// TwinCAT 3 PLC project txi_hxr_optics
// Title: lcls-plc-txi-hxr-optics
// Company: SLAC
// ProjectVersion: 1.0.0
// ProgramVersion: 3.1.4022.7
// libraries:
//   lcls-twincat-motion, * (SLAC)
//   lcls-twincat-optics, * (SLAC)
//   PMPS, * (SLAC - LCLS)
//   Tc2_Standard, * (Beckhoff Automation GmbH)
//   Tc2_System, * (Beckhoff Automation GmbH)
//   Tc3_Module, * (Beckhoff Automation GmbH)
// project tree:
//   GVLs/ GVL_MR1L1_Constants.TcGVL, GVL_PMPS.TcGVL, Main.TcGVL
//   Version/ Global_Version.TcGVL
//   / PlcTask.TcTTO
//   POUs/ PRG_1_PlcTask.TcPOU, PRG_2_PMPS_POST.TcPOU, PRG_MR1L1_HOMS.TcPOU
// real-time tasks:
//   TASK PlcTask: cycle T#10ms, priority 20, ADS port 350
// motion (NC):
//   TASK NC-Task 1 SAF: cycle T#2ms, priority 4, ADS port 501
//   TASK NC-Task 1 SVB: cycle T#10ms, priority 8, ADS port 511
//   AXIS Axis 1 MR1L1-HOMS-YUP (id 1)
//     General: UnitName=um
//     Dynamic: Acceleration=5050, Deceleration=5050, Jerk=5100500, DelayTime=0.008
//     Velo: SlowManual=60, FastManual=90, Maximum=500
//     OtherSettings: AllowMotionCmdToSlave=true
//     encoder EncType=29
//       EncPara: ScaleFactorNumerator=1, ScaleFactorDenominator=1000, MaxCount=#xffffffff
//         SoftEndMaxControl: Enable=true, Range=121500
//         Inc: RefSoftSyncMask=#x0000ffff
//     drive DrvType=24
//       DrvPara: Inverse=true
//         Analog: VeloReferenz=500, ScaleFactorActTorque=0.1
//         TimeComp: TaskDelayCycles=1
//     controller CtrType=3
//       CtrPara: PriorControlFactor=1
//         PosDiffControl: Range=50, Time=0.2
//         PID: PosTn=0.005, PosIOutputLimit=0.0001, PosDOutputLimit=0, PosIDisableWhenMoving=true, DeadBandPosition=0.001
//         Observer: BandWidth=20
//   AXIS Axis 2 MR1L1-HOMS-YDWN (id 2)
//     General: UnitName=um
//     Dynamic: Acceleration=5050, Deceleration=5050, Jerk=5100500, DelayTime=0.008
//     Velo: SlowManual=60, FastManual=90, Maximum=500
//     OtherSettings: AllowMotionCmdToSlave=true
//     encoder EncType=29
//       EncPara: ScaleFactorNumerator=1, ScaleFactorDenominator=1000, MaxCount=#xffffffff
//         Inc: RefSoftSyncMask=#x0000ffff
//     drive DrvType=24
//       DrvPara: Inverse=true
//         Analog: VeloReferenz=500, ScaleFactorActTorque=0.1
//         TimeComp: TaskDelayCycles=1
//     controller CtrType=3
//       CtrPara: PriorControlFactor=1
//         PosDiffControl: Range=50, Time=0.2
//         PID: PosTn=0.005, PosIOutputLimit=0.0001, PosDOutputLimit=0, PosIDisableWhenMoving=true, DeadBandPosition=0.001
//         Observer: BandWidth=20
//   AXIS Axis 3 MR1L1-HOMS-XUP (id 3)
//     General: UnitName=um
//     Dynamic: Acceleration=1000, Deceleration=1000, Jerk=5000, DelayTime=0.008
//     Velo: FastManual=150, Maximum=150
//     OtherSettings: AllowMotionCmdToSlave=true
//     encoder EncType=29
//       EncPara: ScaleFactorNumerator=0.001, MaxCount=#xffffffff
//         Inc: RefSoftSyncMask=#x0000ffff
//     drive DrvType=24
//       DrvPara: Inverse=true
//         Analog: VeloReferenz=625, ScaleFactorActTorque=0.1
//         TimeComp: TaskDelayCycles=1
//     controller CtrType=1
//       CtrPara: PriorControlFactor=1
//         PosDiffControl: Range=50
//         Observer: BandWidth=20
//   AXIS Axis 4 MR1L1-HOMS-XDWN (id 4)
//     General: UnitName=um
//     Dynamic: Acceleration=1000, Deceleration=1000, Jerk=5000, DelayTime=0.008
//     Velo: FastManual=150, Maximum=150
//     OtherSettings: AllowMotionCmdToSlave=true
//     encoder EncType=29
//       EncPara: ScaleFactorNumerator=0.001, MaxCount=#xffffffff
//         Inc: RefSoftSyncMask=#x0000ffff
//     drive DrvType=24
//       Analog: VeloReferenz=625, ScaleFactorActTorque=0.1
//       TimeComp: TaskDelayCycles=1
//     controller CtrType=1
//       CtrPara: PriorControlFactor=1
//         PosDiffControl: Range=50
//         Observer: BandWidth=20
//   AXIS Axis 5 MR1L1-HOMS-PITCH (id 5)
//     General: UnitName=urad
//     Dynamic: AccelerationMaximum=7042, Acceleration=7000, Deceleration=14000, DelayTime=0.008, VeloJumpFactor=2000
//     Velo: SlowManual=30, FastManual=50, Maximum=400
//     MotionControl: Time=0.1
//     TargetPosControl: Time=2
//     OtherSettings: AllowMotionCmdToSlave=true, AllowMotionCmdToExtSetGenAxis=true, PulseDistancePos=100
//     encoder EncType=29
//       EncPara: ScaleFactorNumerator=0.00556, MaxCount=#xffffffff
//         Inc: RefSoftSyncMask=#x0000ffff
//     drive DrvType=24
//       DrvPara: Inverse=true
//         Analog: VeloReferenz=550.176
//         TimeComp: TaskDelayCycles=1
//     controller CtrType=3
//       CtrPara: PriorControlFactor=1
//         PosDiffControl: Range=10, Time=0.2
//         PID: PosKp=8, PosTn=0.0005, PosIOutputLimit=5e-05, PosDOutputLimit=0, DeadBandPosition=0.1
//         Observer: BandWidth=20
// I/O:
//   DEVICE Device 1 (EtherCAT), AmsNetId 172.21.136.43.2.1
//     Term 1 (EK1200) [EK1200-5000 EtherCAT Power supply (2A E-Bus)]
//       PMPS_FFO
//       License (6070)
//       PMPS_PRE [EL6695 EtherCAT Bridge terminal (Primary)]
//       PLC Junction 1 (EK1122) [EK1122 2 port EtherCAT junction]
//         X1 MR1L1 (EK1100) [EK1100 EtherCAT Coupler (2A E-Bus)]
//           Term 8 (EL9410)
//           MR1L1-EL7047-E01 [EL7047 1Ch. Stepper motor output stage (50V, 5A)]
//           MR1L1-EL7047-E02 [EL7047 1Ch. Stepper motor output stage (50V, 5A)]
//           MR1L1-EL7047-E03 [EL7047 1Ch. Stepper motor output stage (50V, 5A)]
//           MR1L1-EL7047-E04 [EL7047 1Ch. Stepper motor output stage (50V, 5A)]
//           MR1L1-EL7047-E05 [EL7047 1Ch. Stepper motor output stage (50V, 5A)]
//           MR1L1-EL5042-E06 [EL5042 2Ch. BiSS-C Encoder]
//           MR1L1-EL5042-E07 [EL5042 2Ch. BiSS-C Encoder]
//           MR1L1-EL5042-E08 [EL5042 2Ch. BiSS-C Encoder]
//           MR1L1-EL6001-E09 [EL6001 Interface (RS232)]
//           MR1L1-EL3054-E10 [EL3054 4Ch. Ana. Input 4-20mA]
//           MR1L1-EL3202-0010-E11 [EL3202-0010 2Ch. Ana. Input PT100 (RTD), High Precision]
//           MR1L1-EL3202-0010-E12 [EL3202-0010 2Ch. Ana. Input PT100 (RTD), High Precision]
//           MR1L1-EL1004-E13
//           MR1L1-EL2004-E14 [EL2004 4Ch. Dig. Output 24V, 0.5A]
//           Term 19 (EL9011) [EL9011 End Terminal]
// variable links:
//   Axes/Axis 1 MR1L1-HOMS-YUP <-> Device 1 (EtherCAT)/Term 1 (EK1200)/PLC Junction 1 (EK1122)/X1 MR1L1 (EK1100)/MR1L1-EL5042-E06
//     Enc/Inputs/In/nComState @bit 1 <-> WcState/InputToggle
//     Enc/Inputs/In/nComState <-> WcState/WcState
//     Enc/Inputs/In/nDataIn1 <-> FB Inputs Channel 1/Position
//     Enc/Inputs/In/nState1 @bit 12 <-> FB Inputs Channel 1/Status/Diag
//     Enc/Inputs/In/nState1 @bit 1 <-> FB Inputs Channel 1/Status/Error
//     Enc/Inputs/In/nState1 @bit 14 <-> FB Inputs Channel 1/Status/Input cycle counter
//     Enc/Inputs/In/nState1 @bit 2 <-> FB Inputs Channel 1/Status/Ready
//     Enc/Inputs/In/nState1 @bit 13 <-> FB Inputs Channel 1/Status/TxPDO State
//     Enc/Inputs/In/nState1 <-> FB Inputs Channel 1/Status/Warning
//   Axes/Axis 1 MR1L1-HOMS-YUP <-> Device 1 (EtherCAT)/Term 1 (EK1200)/PLC Junction 1 (EK1122)/X1 MR1L1 (EK1100)/MR1L1-EL7047-E01
//     Drive/Inputs/In/nState1 @bit 3 <-> STM Status/Status/Error
//     Drive/Inputs/In/nState1 @bit 7 <-> STM Status/Status/Motor stall
//     Drive/Inputs/In/nState1 @bit 5 <-> STM Status/Status/Moving negative
//     Drive/Inputs/In/nState1 @bit 4 <-> STM Status/Status/Moving positive
//     Drive/Inputs/In/nState1 @bit 1 <-> STM Status/Status/Ready
//     Drive/Inputs/In/nState1 <-> STM Status/Status/Ready to enable
//     Drive/Inputs/In/nState1 @bit 6 <-> STM Status/Status/Torque reduced
//     Drive/Inputs/In/nState1 @bit 2 <-> STM Status/Status/Warning
//     Drive/Inputs/In/nState2 @bit 3 <-> STM Status/Status/Digital input 1
//     Drive/Inputs/In/nState2 @bit 4 <-> STM Status/Status/Digital input 2
//     Drive/Inputs/In/nState2 @bit 5 <-> STM Status/Status/Sync error
//     Drive/Inputs/In/nState2 @bit 7 <-> STM Status/Status/TxPDO Toggle
//     Drive/Inputs/In/nState4 @bit 1 <-> WcState/InputToggle
//     Drive/Inputs/In/nState4 <-> WcState/WcState
//     Drive/Outputs/Out/nCtrl1 <-> STM Control/Control/Enable
//     Drive/Outputs/Out/nCtrl1 @bit 2 <-> STM Control/Control/Reduce torque
//     Drive/Outputs/Out/nCtrl1 @bit 1 <-> STM Control/Control/Reset
//     Drive/Outputs/Out/nCtrl2 @bit 3 <-> STM Control/Control/Digital output 1
//     Drive/Outputs/Out/nDataOut2[0] <-> STM Velocity/Velocity
//   Axes/Axis 2 MR1L1-HOMS-YDWN <-> Device 1 (EtherCAT)/Term 1 (EK1200)/PLC Junction 1 (EK1122)/X1 MR1L1 (EK1100)/MR1L1-EL5042-E06
//     Enc/Inputs/In/nComState @bit 1 <-> WcState/InputToggle
//     Enc/Inputs/In/nComState <-> WcState/WcState
//     Enc/Inputs/In/nDataIn1 <-> FB Inputs Channel 2/Position
//     Enc/Inputs/In/nState1 @bit 12 <-> FB Inputs Channel 2/Status/Diag
//     Enc/Inputs/In/nState1 @bit 1 <-> FB Inputs Channel 2/Status/Error
//     Enc/Inputs/In/nState1 @bit 14 <-> FB Inputs Channel 2/Status/Input cycle counter
//     Enc/Inputs/In/nState1 @bit 2 <-> FB Inputs Channel 2/Status/Ready
//     Enc/Inputs/In/nState1 @bit 13 <-> FB Inputs Channel 2/Status/TxPDO State
//     Enc/Inputs/In/nState1 <-> FB Inputs Channel 2/Status/Warning
//   Axes/Axis 2 MR1L1-HOMS-YDWN <-> Device 1 (EtherCAT)/Term 1 (EK1200)/PLC Junction 1 (EK1122)/X1 MR1L1 (EK1100)/MR1L1-EL7047-E02
//     Drive/Inputs/In/nState1 @bit 3 <-> STM Status/Status/Error
//     Drive/Inputs/In/nState1 @bit 7 <-> STM Status/Status/Motor stall
//     Drive/Inputs/In/nState1 @bit 5 <-> STM Status/Status/Moving negative
//     Drive/Inputs/In/nState1 @bit 4 <-> STM Status/Status/Moving positive
//     Drive/Inputs/In/nState1 @bit 1 <-> STM Status/Status/Ready
//     Drive/Inputs/In/nState1 <-> STM Status/Status/Ready to enable
//     Drive/Inputs/In/nState1 @bit 6 <-> STM Status/Status/Torque reduced
//     Drive/Inputs/In/nState1 @bit 2 <-> STM Status/Status/Warning
//     Drive/Inputs/In/nState2 @bit 3 <-> STM Status/Status/Digital input 1
//     Drive/Inputs/In/nState2 @bit 4 <-> STM Status/Status/Digital input 2
//     Drive/Inputs/In/nState2 @bit 5 <-> STM Status/Status/Sync error
//     Drive/Inputs/In/nState2 @bit 7 <-> STM Status/Status/TxPDO Toggle
//     Drive/Inputs/In/nState4 @bit 1 <-> WcState/InputToggle
//     Drive/Inputs/In/nState4 <-> WcState/WcState
//     Drive/Outputs/Out/nCtrl1 <-> STM Control/Control/Enable
//     Drive/Outputs/Out/nCtrl1 @bit 2 <-> STM Control/Control/Reduce torque
//     Drive/Outputs/Out/nCtrl1 @bit 1 <-> STM Control/Control/Reset
//     Drive/Outputs/Out/nCtrl2 @bit 3 <-> STM Control/Control/Digital output 1
//     Drive/Outputs/Out/nDataOut2[0] <-> STM Velocity/Velocity
//   Axes/Axis 3 MR1L1-HOMS-XUP <-> Device 1 (EtherCAT)/Term 1 (EK1200)/PLC Junction 1 (EK1122)/X1 MR1L1 (EK1100)/MR1L1-EL5042-E07
//     Enc/Inputs/In/nComState @bit 1 <-> WcState/InputToggle
//     Enc/Inputs/In/nComState <-> WcState/WcState
//     Enc/Inputs/In/nDataIn1 <-> FB Inputs Channel 1/Position
//     Enc/Inputs/In/nState1 @bit 12 <-> FB Inputs Channel 1/Status/Diag
//     Enc/Inputs/In/nState1 @bit 1 <-> FB Inputs Channel 1/Status/Error
//     Enc/Inputs/In/nState1 @bit 14 <-> FB Inputs Channel 1/Status/Input cycle counter
//     Enc/Inputs/In/nState1 @bit 2 <-> FB Inputs Channel 1/Status/Ready
//     Enc/Inputs/In/nState1 @bit 13 <-> FB Inputs Channel 1/Status/TxPDO State
//     Enc/Inputs/In/nState1 <-> FB Inputs Channel 1/Status/Warning
//   Axes/Axis 3 MR1L1-HOMS-XUP <-> Device 1 (EtherCAT)/Term 1 (EK1200)/PLC Junction 1 (EK1122)/X1 MR1L1 (EK1100)/MR1L1-EL7047-E03
//     Drive/Inputs/In/nState1 @bit 3 <-> STM Status/Status/Error
//     Drive/Inputs/In/nState1 @bit 7 <-> STM Status/Status/Motor stall
//     Drive/Inputs/In/nState1 @bit 5 <-> STM Status/Status/Moving negative
//     Drive/Inputs/In/nState1 @bit 4 <-> STM Status/Status/Moving positive
//     Drive/Inputs/In/nState1 @bit 1 <-> STM Status/Status/Ready
//     Drive/Inputs/In/nState1 <-> STM Status/Status/Ready to enable
//     Drive/Inputs/In/nState1 @bit 6 <-> STM Status/Status/Torque reduced
//     Drive/Inputs/In/nState1 @bit 2 <-> STM Status/Status/Warning
//     Drive/Inputs/In/nState2 @bit 3 <-> STM Status/Status/Digital input 1
//     Drive/Inputs/In/nState2 @bit 4 <-> STM Status/Status/Digital input 2
//     Drive/Inputs/In/nState2 @bit 5 <-> STM Status/Status/Sync error
//     Drive/Inputs/In/nState2 @bit 7 <-> STM Status/Status/TxPDO Toggle
//     Drive/Inputs/In/nState4 @bit 1 <-> WcState/InputToggle
//     Drive/Inputs/In/nState4 <-> WcState/WcState
//     Drive/Outputs/Out/nCtrl1 <-> STM Control/Control/Enable
//     Drive/Outputs/Out/nCtrl1 @bit 2 <-> STM Control/Control/Reduce torque
//     Drive/Outputs/Out/nCtrl1 @bit 1 <-> STM Control/Control/Reset
//     Drive/Outputs/Out/nCtrl2 @bit 3 <-> STM Control/Control/Digital output 1
//     Drive/Outputs/Out/nDataOut2[0] <-> STM Velocity/Velocity
//   Axes/Axis 4 MR1L1-HOMS-XDWN <-> Device 1 (EtherCAT)/Term 1 (EK1200)/PLC Junction 1 (EK1122)/X1 MR1L1 (EK1100)/MR1L1-EL5042-E07
//     Enc/Inputs/In/nComState @bit 1 <-> WcState/InputToggle
//     Enc/Inputs/In/nComState <-> WcState/WcState
//     Enc/Inputs/In/nDataIn1 <-> FB Inputs Channel 2/Position
//     Enc/Inputs/In/nState1 @bit 12 <-> FB Inputs Channel 2/Status/Diag
//     Enc/Inputs/In/nState1 @bit 1 <-> FB Inputs Channel 2/Status/Error
//     Enc/Inputs/In/nState1 @bit 14 <-> FB Inputs Channel 2/Status/Input cycle counter
//     Enc/Inputs/In/nState1 @bit 2 <-> FB Inputs Channel 2/Status/Ready
//     Enc/Inputs/In/nState1 @bit 13 <-> FB Inputs Channel 2/Status/TxPDO State
//     Enc/Inputs/In/nState1 <-> FB Inputs Channel 2/Status/Warning
//   Axes/Axis 4 MR1L1-HOMS-XDWN <-> Device 1 (EtherCAT)/Term 1 (EK1200)/PLC Junction 1 (EK1122)/X1 MR1L1 (EK1100)/MR1L1-EL7047-E04
//     Drive/Inputs/In/nState1 @bit 3 <-> STM Status/Status/Error
//     Drive/Inputs/In/nState1 @bit 7 <-> STM Status/Status/Motor stall
//     Drive/Inputs/In/nState1 @bit 5 <-> STM Status/Status/Moving negative
//     Drive/Inputs/In/nState1 @bit 4 <-> STM Status/Status/Moving positive
//     Drive/Inputs/In/nState1 @bit 1 <-> STM Status/Status/Ready
//     Drive/Inputs/In/nState1 <-> STM Status/Status/Ready to enable
//     Drive/Inputs/In/nState1 @bit 6 <-> STM Status/Status/Torque reduced
//     Drive/Inputs/In/nState1 @bit 2 <-> STM Status/Status/Warning
//     Drive/Inputs/In/nState2 @bit 3 <-> STM Status/Status/Digital input 1
//     Drive/Inputs/In/nState2 @bit 4 <-> STM Status/Status/Digital input 2
//     Drive/Inputs/In/nState2 @bit 5 <-> STM Status/Status/Sync error
//     Drive/Inputs/In/nState2 @bit 7 <-> STM Status/Status/TxPDO Toggle
//     Drive/Inputs/In/nState4 @bit 1 <-> WcState/InputToggle
//     Drive/Inputs/In/nState4 <-> WcState/WcState
//     Drive/Outputs/Out/nCtrl1 <-> STM Control/Control/Enable
//     Drive/Outputs/Out/nCtrl1 @bit 2 <-> STM Control/Control/Reduce torque
//     Drive/Outputs/Out/nCtrl1 @bit 1 <-> STM Control/Control/Reset
//     Drive/Outputs/Out/nCtrl2 @bit 3 <-> STM Control/Control/Digital output 1
//     Drive/Outputs/Out/nDataOut2[0] <-> STM Velocity/Velocity
//   Axes/Axis 5 MR1L1-HOMS-PITCH <-> Device 1 (EtherCAT)/Term 1 (EK1200)/PLC Junction 1 (EK1122)/X1 MR1L1 (EK1100)/MR1L1-EL5042-E08
//     Enc/Inputs/In/nComState @bit 1 <-> WcState/InputToggle
//     Enc/Inputs/In/nComState <-> WcState/WcState
//     Enc/Inputs/In/nDataIn1 <-> FB Inputs Channel 1/Position
//     Enc/Inputs/In/nState1 @bit 12 <-> FB Inputs Channel 1/Status/Diag
//     Enc/Inputs/In/nState1 @bit 1 <-> FB Inputs Channel 1/Status/Error
//     Enc/Inputs/In/nState1 @bit 14 <-> FB Inputs Channel 1/Status/Input cycle counter
//     Enc/Inputs/In/nState1 @bit 2 <-> FB Inputs Channel 1/Status/Ready
//     Enc/Inputs/In/nState1 @bit 13 <-> FB Inputs Channel 1/Status/TxPDO State
//     Enc/Inputs/In/nState1 <-> FB Inputs Channel 1/Status/Warning
//   Axes/Axis 5 MR1L1-HOMS-PITCH <-> Device 1 (EtherCAT)/Term 1 (EK1200)/PLC Junction 1 (EK1122)/X1 MR1L1 (EK1100)/MR1L1-EL7047-E05
//     Drive/Inputs/In/nState1 @bit 3 <-> STM Status/Status/Error
//     Drive/Inputs/In/nState1 @bit 7 <-> STM Status/Status/Motor stall
//     Drive/Inputs/In/nState1 @bit 5 <-> STM Status/Status/Moving negative
//     Drive/Inputs/In/nState1 @bit 4 <-> STM Status/Status/Moving positive
//     Drive/Inputs/In/nState1 @bit 1 <-> STM Status/Status/Ready
//     Drive/Inputs/In/nState1 <-> STM Status/Status/Ready to enable
//     Drive/Inputs/In/nState1 @bit 6 <-> STM Status/Status/Torque reduced
//     Drive/Inputs/In/nState1 @bit 2 <-> STM Status/Status/Warning
//     Drive/Inputs/In/nState2 @bit 3 <-> STM Status/Status/Digital input 1
//     Drive/Inputs/In/nState2 @bit 4 <-> STM Status/Status/Digital input 2
//     Drive/Inputs/In/nState2 @bit 5 <-> STM Status/Status/Sync error
//     Drive/Inputs/In/nState2 @bit 7 <-> STM Status/Status/TxPDO Toggle
//     Drive/Inputs/In/nState4 @bit 1 <-> WcState/InputToggle
//     Drive/Inputs/In/nState4 <-> WcState/WcState
//     Drive/Outputs/Out/nCtrl1 <-> STM Control/Control/Enable
//     Drive/Outputs/Out/nCtrl1 @bit 2 <-> STM Control/Control/Reduce torque
//     Drive/Outputs/Out/nCtrl1 @bit 1 <-> STM Control/Control/Reset
//     Drive/Outputs/Out/nCtrl2 @bit 3 <-> STM Control/Control/Digital output 1
//     Drive/Outputs/Out/nDataOut2[0] <-> STM Velocity/Velocity
//   txi_hxr_optics Instance <-> Device 1 (EtherCAT)/Term 1 (EK1200)/PLC Junction 1 (EK1122)/X1 MR1L1 (EK1100)/MR1L1-EL1004-E13
//     PlcTask Inputs/PRG_MR1L1_HOMS.MR1L1.fbRunHOMS.bSTOEnable1 <-> Channel 1/Input
//     PlcTask Inputs/PRG_MR1L1_HOMS.MR1L1.fbRunHOMS.bSTOEnable2 <-> Channel 2/Input
//   txi_hxr_optics Instance <-> Device 1 (EtherCAT)/Term 1 (EK1200)/PLC Junction 1 (EK1122)/X1 MR1L1 (EK1100)/MR1L1-EL2004-E14
//     PlcTask Outputs/PRG_MR1L1_HOMS.bActivateVarCool <-> Channel 1/Output
//   txi_hxr_optics Instance <-> Device 1 (EtherCAT)/Term 1 (EK1200)/PLC Junction 1 (EK1122)/X1 MR1L1 (EK1100)/MR1L1-EL3054-E10
//     PlcTask Inputs/PRG_MR1L1_HOMS.fbCoolingPanel.fbFlow_1.iRaw <-> AI Standard Channel 1/Value
//     PlcTask Inputs/PRG_MR1L1_HOMS.fbCoolingPanel.fbFlow_2.iRaw <-> AI Standard Channel 2/Value
//     PlcTask Inputs/PRG_MR1L1_HOMS.fbCoolingPanel.fbPress_1.iRaw <-> AI Standard Channel 3/Value
//   txi_hxr_optics Instance <-> Device 1 (EtherCAT)/Term 1 (EK1200)/PLC Junction 1 (EK1122)/X1 MR1L1 (EK1100)/MR1L1-EL5042-E06
//     PlcTask Inputs/Main.M1.nRawEncoderULINT <-> FB Inputs Channel 1/Position
//     PlcTask Inputs/Main.M2.nRawEncoderULINT <-> FB Inputs Channel 2/Position
//     PlcTask Inputs/PRG_MR1L1_HOMS.MR1L1.fbRunHOMS.stYdwnEnc/Count <-> FB Inputs Channel 2/Position
//     PlcTask Inputs/PRG_MR1L1_HOMS.MR1L1.fbRunHOMS.stYupEnc/Count <-> FB Inputs Channel 1/Position
//     PlcTask Inputs/PRG_MR1L1_HOMS.bMR1L1_Y_ENC_Ready <-> FB Inputs Channel 1/Status/Ready
//     PlcTask Inputs/PRG_MR1L1_HOMS.bMR1L1_Y_ENC_TxPDO <-> FB Inputs Channel 1/Status/TxPDO State
//   txi_hxr_optics Instance <-> Device 1 (EtherCAT)/Term 1 (EK1200)/PLC Junction 1 (EK1122)/X1 MR1L1 (EK1100)/MR1L1-EL5042-E07
//     PlcTask Inputs/Main.M3.nRawEncoderULINT <-> FB Inputs Channel 1/Position
//     PlcTask Inputs/Main.M4.nRawEncoderULINT <-> FB Inputs Channel 2/Position
//     PlcTask Inputs/PRG_MR1L1_HOMS.MR1L1.fbRunHOMS.stXdwnEnc/Count <-> FB Inputs Channel 2/Position
//     PlcTask Inputs/PRG_MR1L1_HOMS.MR1L1.fbRunHOMS.stXupEnc/Count <-> FB Inputs Channel 1/Position
//   txi_hxr_optics Instance <-> Device 1 (EtherCAT)/Term 1 (EK1200)/PLC Junction 1 (EK1122)/X1 MR1L1 (EK1100)/MR1L1-EL5042-E08
//     PlcTask Inputs/Main.M5.nRawEncoderULINT <-> FB Inputs Channel 1/Position
//   txi_hxr_optics Instance <-> Device 1 (EtherCAT)/Term 1 (EK1200)/PLC Junction 1 (EK1122)/X1 MR1L1 (EK1100)/MR1L1-EL7047-E01
//     PlcTask Inputs/Main.M1.bLimitBackwardEnable <-> STM Status/Status/Digital input 2
//     PlcTask Inputs/Main.M1.bLimitForwardEnable <-> STM Status/Status/Digital input 1
//   txi_hxr_optics Instance <-> Device 1 (EtherCAT)/Term 1 (EK1200)/PLC Junction 1 (EK1122)/X1 MR1L1 (EK1100)/MR1L1-EL7047-E02
//     PlcTask Inputs/Main.M2.bLimitBackwardEnable <-> STM Status/Status/Digital input 2
//     PlcTask Inputs/Main.M2.bLimitForwardEnable <-> STM Status/Status/Digital input 1
//   txi_hxr_optics Instance <-> Device 1 (EtherCAT)/Term 1 (EK1200)/PLC Junction 1 (EK1122)/X1 MR1L1 (EK1100)/MR1L1-EL7047-E03
//     PlcTask Inputs/Main.M3.bLimitBackwardEnable <-> STM Status/Status/Digital input 2
//     PlcTask Inputs/Main.M3.bLimitForwardEnable <-> STM Status/Status/Digital input 1
//   txi_hxr_optics Instance <-> Device 1 (EtherCAT)/Term 1 (EK1200)/PLC Junction 1 (EK1122)/X1 MR1L1 (EK1100)/MR1L1-EL7047-E04
//     PlcTask Inputs/Main.M4.bLimitBackwardEnable <-> STM Status/Status/Digital input 2
//     PlcTask Inputs/Main.M4.bLimitForwardEnable <-> STM Status/Status/Digital input 1
//   txi_hxr_optics Instance <-> Device 1 (EtherCAT)/Term 1 (EK1200)/PLC Junction 1 (EK1122)/X1 MR1L1 (EK1100)/MR1L1-EL7047-E05
//     PlcTask Inputs/Main.M5.bLimitBackwardEnable <-> STM Status/Status/Digital input 2
//     PlcTask Inputs/Main.M5.bLimitForwardEnable <-> STM Status/Status/Digital input 1
//   txi_hxr_optics Instance <-> Device 1 (EtherCAT)/Term 1 (EK1200)/PMPS_FFO
//     PlcTask Outputs/GVL_PMPS.fbFastFaultOutput1.q_xFastFaultOut <-> Channel 1/Output
//   txi_hxr_optics Instance <-> Device 1 (EtherCAT)/Term 1 (EK1200)/PMPS_PRE
//     PlcTask Inputs/PRG_2_PMPS_POST.fbArbiterIO.i_stCurrentBP <-> IO Inputs/CurrentBP
//     PlcTask Inputs/PRG_2_PMPS_POST.fbArbiterIO.xTxPDO_state <-> SYNC Inputs/TxPDO state
//     PlcTask Inputs/PRG_2_PMPS_POST.fbArbiterIO.xTxPDO_toggle <-> SYNC Inputs/TxPDO toggle
//     PlcTask Outputs/PRG_2_PMPS_POST.fbArbiterIO.q_stRequestedBP <-> IO Outputs/RequestedBP
//     PlcTask Outputs/PRG_MR1L1_HOMS.nMR1L1_Y_ENC_PMPS <-> IO Outputs/MR1L1_Y_ENC
//   txi_hxr_optics Instance <-> NC-Task 1 SAF/Axes/Axis 1 MR1L1-HOMS-YUP
//     PlcTask Inputs/Main.M1.Axis.NcToPlc <-> Outputs/ToPlc
//     PlcTask Outputs/Main.M1.Axis.PlcToNc <-> Inputs/FromPlc
//   txi_hxr_optics Instance <-> NC-Task 1 SAF/Axes/Axis 2 MR1L1-HOMS-YDWN
//     PlcTask Inputs/Main.M2.Axis.NcToPlc <-> Outputs/ToPlc
//     PlcTask Outputs/Main.M2.Axis.PlcToNc <-> Inputs/FromPlc
//   txi_hxr_optics Instance <-> NC-Task 1 SAF/Axes/Axis 3 MR1L1-HOMS-XUP
//     PlcTask Inputs/Main.M3.Axis.NcToPlc <-> Outputs/ToPlc
//     PlcTask Outputs/Main.M3.Axis.PlcToNc <-> Inputs/FromPlc
//   txi_hxr_optics Instance <-> NC-Task 1 SAF/Axes/Axis 4 MR1L1-HOMS-XDWN
//     PlcTask Inputs/Main.M4.Axis.NcToPlc <-> Outputs/ToPlc
//     PlcTask Outputs/Main.M4.Axis.PlcToNc <-> Inputs/FromPlc
//   txi_hxr_optics Instance <-> NC-Task 1 SAF/Axes/Axis 5 MR1L1-HOMS-PITCH
//     PlcTask Inputs/Main.M5.Axis.NcToPlc <-> Outputs/ToPlc
//     PlcTask Outputs/Main.M5.Axis.PlcToNc <-> Inputs/FromPlc

CONFIGURATION txi_hxr_optics
    RESOURCE PLC ON TwinCAT3
        TASK PlcTask(INTERVAL := T#10ms, PRIORITY := 20);
        PROGRAM PRG_1_PlcTask WITH PlcTask : PRG_1_PlcTask;
    END_RESOURCE
END_CONFIGURATION

// ---- GVLs/GVL_MR1L1_Constants.TcGVL
{attribute 'qualified_only'}
VAR_GLOBAL
    nYUP_ENC_REF : ULINT := 108558460;
    nYDWN_ENC_REF : ULINT := 108761210;
    nXUP_ENC_REF : ULINT := 20664670;
    nXDWN_ENC_REF : ULINT := 20133000;
END_VAR

// ---- Version/Global_Version.TcGVL
{attribute 'TcGenerated'}
{attribute 'no-analysis'}
{attribute 'linkalways'}
// This function has been automatically generated from the project information.
VAR_GLOBAL CONSTANT
    {attribute 'const_non_replaced'}
    stLibVersion_lcls_plc_txi_hxr_optics : ST_LibVersion := (iMajor := 1, iMinor := 0, iBuild := 0, iRevision := 0, nFlags := 1, sVersion := '1.0.0');
END_VAR

// ---- GVLs/GVL_PMPS.TcGVL
{attribute 'qualified_only'}
VAR_GLOBAL
    {attribute 'pytmc' := 'pv: PLC:TXI:LFE:OPTICS:ARB:01'}
    fbArbiter1: FB_Arbiter(1);
    {attribute 'pytmc' := 'pv: PLC:TXI:LFE:OPTICS:ARB:02'}
    fbArbiter2: FB_Arbiter(2);
    {attribute 'pytmc' := 'pv: PLC:TXI:LFE:OPTICS:FFO:01'}
    {attribute 'TcLinkTo' := '.q_xFastFaultOut:=TIIB[PMPS_FFO]^Channel 1^Output'}
    fbFastFaultOutput1: FB_HardwareFFOutput := (bAutoReset := TRUE , i_sNetID:='172.21.42.126.1.1' );
END_VAR

// ---- GVLs/Main.TcGVL
{attribute 'qualified_only'}
VAR_GLOBAL
    {attribute 'TcLinkTo' := '.bLimitForwardEnable:=TIIB[MR1L1-EL7047-E01]^STM Status^Status^Digital input 1;
                              .bLimitBackwardEnable:=TIIB[MR1L1-EL7047-E01]^STM Status^Status^Digital input 2;
                              .nRawEncoderULINT:=TIIB[MR1L1-EL5042-E06]^FB Inputs Channel 1^Position'}
    {attribute 'pytmc' := '
        pv: MR1L1:HOMS:MMS:YUP
    '}
    M1 : ST_MotionStage := (sName:='MR1L1:HOMS:YUP', fVelocity:=100.0, nEnableMode:=ENUM_StageEnableMode.ALWAYS, bPowerSelf:=TRUE);


    {attribute 'TcLinkTo' := '.bLimitForwardEnable:=TIIB[MR1L1-EL7047-E02]^STM Status^Status^Digital input 1;
                              .bLimitBackwardEnable:=TIIB[MR1L1-EL7047-E02]^STM Status^Status^Digital input 2;
                              .nRawEncoderULINT:=TIIB[MR1L1-EL5042-E06]^FB Inputs Channel 2^Position'}
    {attribute 'pytmc' := '
        pv: MR1L1:HOMS:MMS:YDWN
    '}
    M2 : ST_MotionStage := (sName:='MR1L1:HOMS:YDWN', fVelocity:=100.0, nEnableMode:=ENUM_StageEnableMode.ALWAYS, bPowerSelf:=TRUE);

    {attribute 'TcLinkTo' := '.bLimitForwardEnable:=TIIB[MR1L1-EL7047-E03]^STM Status^Status^Digital input 1;
                              .bLimitBackwardEnable:=TIIB[MR1L1-EL7047-E03]^STM Status^Status^Digital input 2;
                              .nRawEncoderULINT:=TIIB[MR1L1-EL5042-E07]^FB Inputs Channel 1^Position'}
    {attribute 'pytmc' := '
        pv: MR1L1:HOMS:MMS:XUP
    '}
    M3 : ST_MotionStage := (sName:='MR1L1:HOMS:XUP', fVelocity:=150.0, nEnableMode:=ENUM_StageEnableMode.ALWAYS, bPowerSelf:=TRUE);



    {attribute 'TcLinkTo' := '.bLimitForwardEnable:=TIIB[MR1L1-EL7047-E04]^STM Status^Status^Digital input 1;
                              .bLimitBackwardEnable:=TIIB[MR1L1-EL7047-E04]^STM Status^Status^Digital input 2;
                              .nRawEncoderULINT:=TIIB[MR1L1-EL5042-E07]^FB Inputs Channel 2^Position'}
    {attribute 'pytmc' := '
        pv: MR1L1:HOMS:MMS:XDWN
    '}
    M4 : ST_MotionStage := (sName:='MR1L1:HOMS:XDWN', fVelocity:=150.0, nEnableMode:=ENUM_StageEnableMode.ALWAYS, bPowerSelf:=TRUE);


    {attribute 'TcLinkTo' := '.bLimitForwardEnable:=TIIB[MR1L1-EL7047-E05]^STM Status^Status^Digital input 1;
                              .bLimitBackwardEnable:=TIIB[MR1L1-EL7047-E05]^STM Status^Status^Digital input 2;
                              .nRawEncoderULINT:=TIIB[MR1L1-EL5042-E08]^FB Inputs Channel 1^Position'}
    {attribute 'pytmc' := '
        pv: MR1L1:HOMS:MMS:PITCH
    '}
    M5 : ST_MotionStage := (sName:='MR1L1:HOMS:PITCH', fVelocity:=150.0, nEnableMode:=ENUM_StageEnableMode.ALWAYS, bPowerSelf:=TRUE);

END_VAR

// ---- POUs/PRG_1_PlcTask.TcPOU
PROGRAM PRG_1_PlcTask
VAR
END_VAR

PRG_MR1L1_HOMS();
PRG_2_PMPS_POST();

END_PROGRAM

// ---- POUs/PRG_MR1L1_HOMS.TcPOU
PROGRAM PRG_MR1L1_HOMS
VAR
    fbMotionStage_m1, fbMotionStage_m2, fbMotionStage_m3, fbMotionStage_m4, fbMotionStage_m5 : FB_MotionStage;

    {attribute 'TcLinkTo' := '.fbRunHOMS.bSTOEnable1:=TIIB[MR1L1-EL1004-E13]^Channel 1^Input;
                              .fbRunHOMS.bSTOEnable2:=TIIB[MR1L1-EL1004-E13]^Channel 2^Input;
                              .fbRunHOMS.stYupEnc.Count:=TIIB[MR1L1-EL5042-E06]^FB Inputs Channel 1^Position;
                              .fbRunHOMS.stYdwnEnc.Count:=TIIB[MR1L1-EL5042-E06]^FB Inputs Channel 2^Position;
                              .fbRunHOMS.stXupEnc.Count:=TIIB[MR1L1-EL5042-E07]^FB Inputs Channel 1^Position;
                              .fbRunHOMS.stXdwnEnc.Count:=TIIB[MR1L1-EL5042-E07]^FB Inputs Channel 2^Position'}
    {attribute 'pytmc' := '
        pv: MR1L1:HOMS
    '}
    MR1L1 : DUT_HOMS;
    // MR1L1 Y Encoder for PMPS Veto Device
    ///////////////////////////////////////
    {attribute 'TcLinkTo' := 'TIIB[PMPS_PRE]^IO Outputs^MR1L1_Y_ENC'}
    nMR1L1_Y_ENC_PMPS AT %Q* : ULINT;
    {attribute 'TcLinkTo' := 'TIIB[MR1L1-EL5042-E06]^FB Inputs Channel 1^Status^Ready'}
    bMR1L1_Y_ENC_Ready AT %I* : BOOL;
    {attribute 'TcLinkTo' := 'TIIB[MR1L1-EL5042-E06]^FB Inputs Channel 1^Status^TxPDO State'}
    bMR1L1_Y_ENC_TxPDO AT %I* : BOOL;
    {attribute 'TcLinkTo' := 'TIIB[MR1L1-EL2004-E14]^Channel 1^Output'}
     {attribute 'pytmc' := '
        pv: MR1L1:HOMS:VCV
        io: io
        field: ZNAM OFF
        field: ONAM ON
    '}
    bActivateVarCool AT %Q* : BOOL;
        // MR1L1 Flow Sensors
    {attribute 'TcLinkTo' := '.fbFlow_1.iRaw := TIIB[MR1L1-EL3054-E10]^AI Standard Channel 1^Value;
                              .fbFlow_2.iRaw := TIIB[MR1L1-EL3054-E10]^AI Standard Channel 2^Value;
                              .fbPress_1.iRaw := TIIB[MR1L1-EL3054-E10]^AI Standard Channel 3^Value
    '}
    {attribute 'pytmc' := '
        pv: MR1L1:HOMS
    '}
    fbCoolingPanel : FB_Axilon_Cooling_2f1p;



END_VAR

// MR1L3 BECKHOFF
MR1L1.fbRunHOMS(stYup:=Main.M1,
               stYdwn:=Main.M2,
               stXup:=Main.M3,
               stXdwn:=Main.M4,
               stPitch:=Main.M5,
               nYupEncRef:=GVL_MR1L1_Constants.nYUP_ENC_REF,
               nYdwnEncRef:=GVL_MR1L1_Constants.nYDWN_ENC_REF,
               nXupEncRef:=GVL_MR1L1_Constants.nXUP_ENC_REF,
               nXdwnEncRef:=GVL_MR1L1_Constants.nXDWN_ENC_REF,
               bExecuteCoupleY:=MR1L1.bExecuteCoupleY,
               bExecuteCoupleX:=MR1L1.bExecuteCoupleX,
               bExecuteDecoupleY:=MR1L1.bExecuteDecoupleY,
               bExecuteDecoupleX:=MR1L1.bExecuteDecoupleX,
               bGantryAlreadyCoupledY=>MR1L1.bGantryAlreadyCoupledY,
               bGantryAlreadyCoupledX=>MR1L1.bGantryAlreadyCoupledX,
               nCurrGantryY=>MR1L1.nCurrGantryY,
               nCurrGantryX=>MR1L1.nCurrGantryX);
// No slave motion through Epics
Main.M2.bExecute := FALSE; // MR1L1-Ydwn
Main.M4.bExecute := FALSE; // MR1L1-Xdwn

fbMotionStage_m1(stMotionStage:=Main.M1);
fbMotionStage_m2(stMotionStage:=Main.M2);
fbMotionStage_m3(stMotionStage:=Main.M3);
fbMotionStage_m4(stMotionStage:=Main.M4);
fbMotionStage_m5(stMotionStage:=Main.M5);

nMR1L1_Y_ENC_PMPS := Main.M1.nRawEncoderULINT;

fbCoolingPanel();

END_PROGRAM

// ---- POUs/PRG_2_PMPS_POST.TcPOU
PROGRAM PRG_2_PMPS_POST
VAR
    fbArbiterIO: FB_SubSysToArbiter_IO;
    fb_vetoArbiter: FB_VetoArbiter;
END_VAR


GVL_PMPS.fbFastFaultOutput1.Execute();

fbArbiterIO(
    Arbiter:=GVL_PMPS.fbArbiter1,
    fbFFHWO:=GVL_PMPS.fbFastFaultOutput1);
//Arb2 in hutch
fb_vetoArbiter(bVeto:= PMPS_GVL.stCurrentBeamParameters.aVetoDevices[PMPS.L_Stopper.ST1L1],
                HigherAuthority := GVL_PMPS.fbArbiter1,
                LowerAuthority := GVL_PMPS.fbArbiter2,
                FFO := GVL_PMPS.fbFastFaultOutput1);

//ff2_ff1_link_optics(
    //io_fbFFHWO := GVL_PMPS.fbFastFaultOutput1,
    //i_xOK :=  GVL_PMPS.fbFastFaultOutput2.q_xFastFaultOut);

//Code for Removing arbitration
GVL_PMPS.fbArbiter1.AddRequest(nReqID := 47, stReqBp := PMPS_GVL.cstFullBeam, sDevName := 'txi-lfe-optics');
GVL_PMPS.fbArbiter2.AddRequest(nReqID := 48, stReqBp := PMPS_GVL.cstFullBeam, sDevName := 'txi-lfe-optics');

//send encoder values for veto

END_PROGRAM
